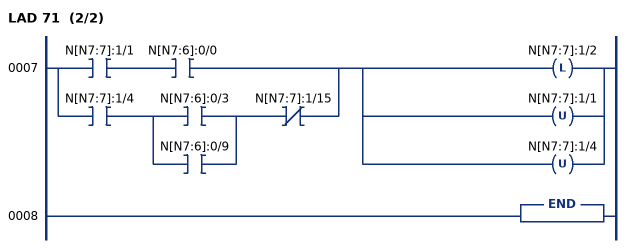
% Rung: 7 %
SOR BST XIC N[N7:7]:1/1 XIC N[N7:6]:0/0 NXB XIC N[N7:7]:1/4 BST XIC N[N7:6]:0/3 NXB XIC N[N7:6]:0/9 BND XIO N[N7:7]:1/15 BND BST OTL N[N7:7]:1/2 NXB OTU N[N7:7]:1/1 NXB OTU N[N7:7]:1/4 BND EOR
% Rung: 8 %
SOR END EOR

LADDER 74
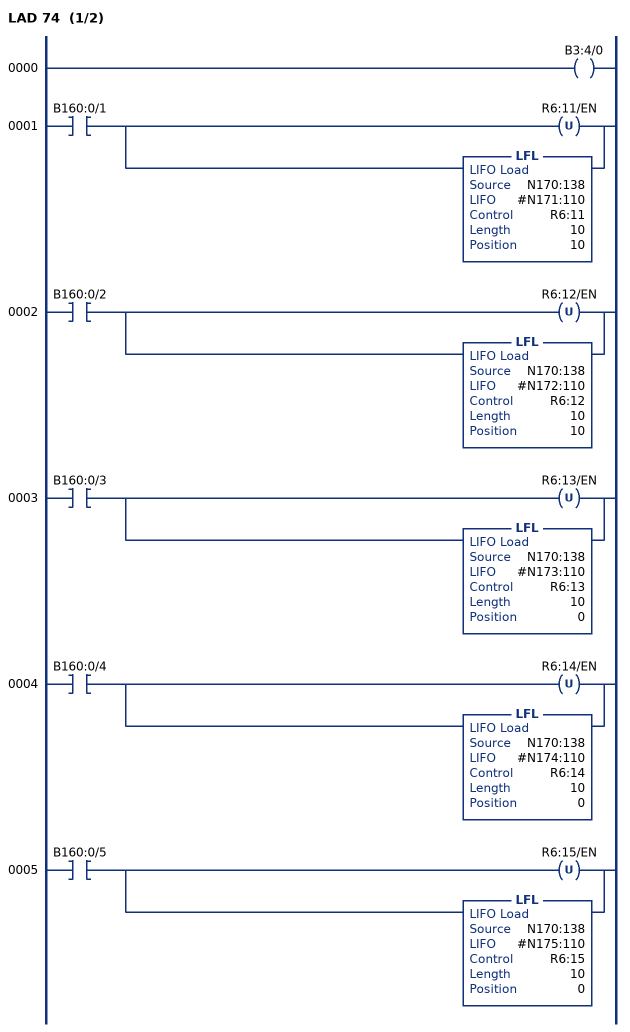
% Rung: 0 %
SOR OTE B3:4/0 EOR
% Rung: 1 %
SOR XIC B160:0/1 BST OTU R6:11/EN NXB LFL N170:138 #N171:110 R6:11 10 10 BND EOR
% Rung: 2 %
SOR XIC B160:0/2 BST OTU R6:12/EN NXB LFL N170:138 #N172:110 R6:12 10 10 BND EOR
% Rung: 3 %
SOR XIC B160:0/3 BST OTU R6:13/EN NXB LFL N170:138 #N173:110 R6:13 10 0 BND EOR
% Rung: 4 %
SOR XIC B160:0/4 BST OTU R6:14/EN NXB LFL N170:138 #N174:110 R6:14 10 0 BND EOR
% Rung: 5 %
SOR XIC B160:0/5 BST OTU R6:15/EN NXB LFL N170:138 #N175:110 R6:15 10 0 BND EOR

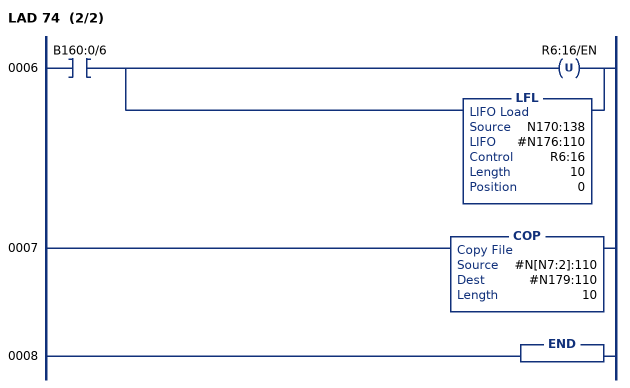
% Rung: 6 %
SOR XIC B160:0/6 BST OTU R6:16/EN NXB LFL N170:138 #N176:110 R6:16 10 0 BND EOR
% Rung: 7 %
SOR COP #N[N7:2]:110 #N179:110 10 EOR
% Rung: 8 %
SOR END EOR

LADDER 75
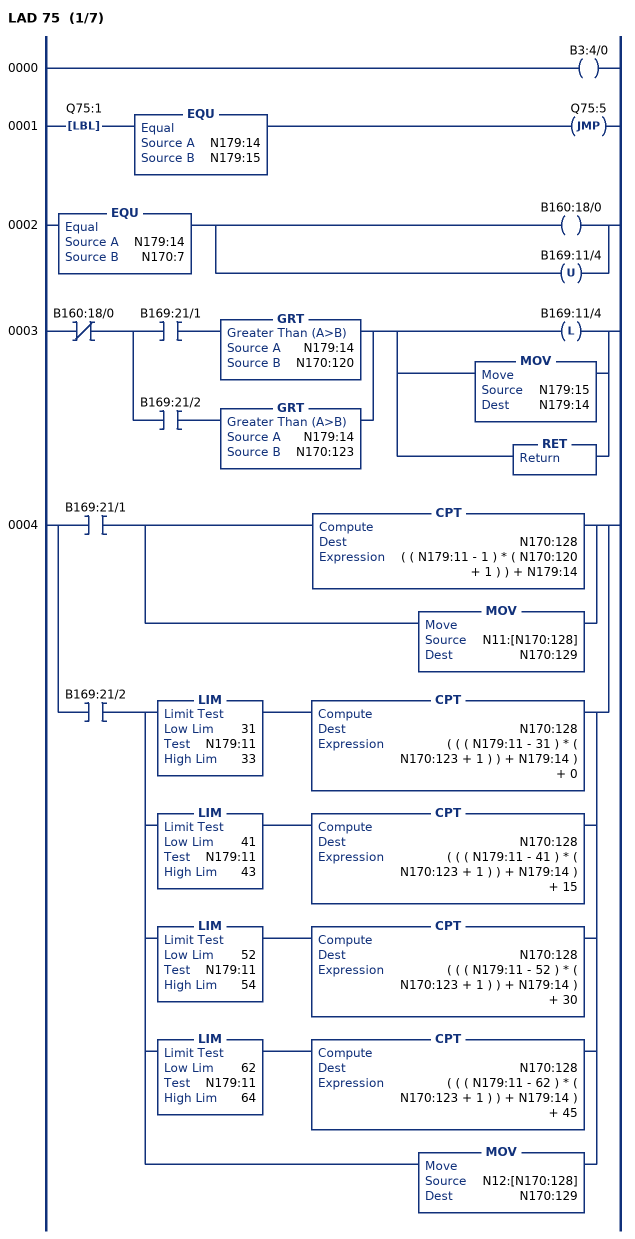
% Rung: 0 %
SOR OTE B3:4/0 EOR
% Rung: 1 %
SOR LBL Q75:1 EQU N179:14 N179:15 JMP Q75:5 EOR
% Rung: 2 %
SOR EQU N179:14 N170:7 BST OTE B160:18/0 NXB OTU B169:11/4 BND EOR
% Rung: 3 %
SOR XIO B160:18/0 BST XIC B169:21/1 GRT N179:14 N170:120 NXB XIC B169:21/2 GRT N179:14 N170:123 BND BST OTL B169:11/4 NXB MOV N179:15 N179:14 NXB RET BND EOR
% Rung: 4 %
SOR BST XIC B169:21/1 BST CPT N170:128 " ( ( N179:11 - 1 ) * ( N170:120 + 1 ) ) + N179:14 " NXB MOV N11:[N170:128] N170:129 BND NXB XIC B169:21/2 BST BST LIM 31 N179:11 33 CPT N170:128 " ( ( ( N179:11 - 31 ) * ( N170:123 + 1 ) ) + N179:14 ) + 0 " NXB LIM 41 N179:11 43 CPT N170:128 " ( ( ( N179:11 - 41 ) * ( N170:123 + 1 ) ) + N179:14 ) + 15 " NXB LIM 52 N179:11 54 CPT N170:128 " ( ( ( N179:11 - 52 ) * ( N170:123 + 1 ) ) + N179:14 ) + 30 " NXB LIM 62 N179:11 64 CPT N170:128 " ( ( ( N179:11 - 62 ) * ( N170:123 + 1 ) ) + N179:14 ) + 45 " BND NXB MOV N12:[N170:128] N170:129 BND BND EOR

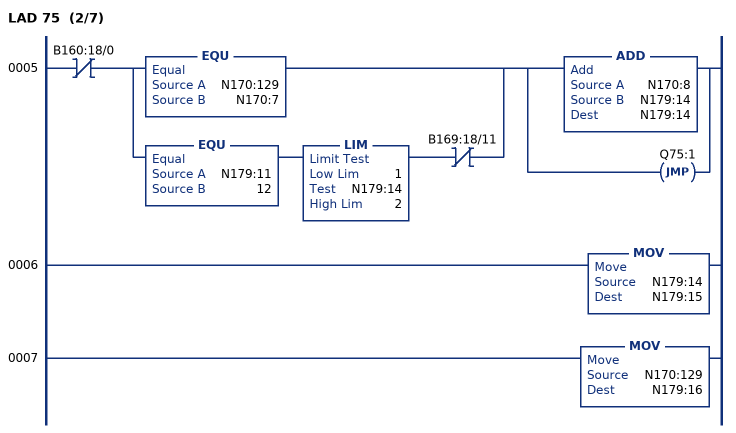
% Rung: 5 %
SOR XIO B160:18/0 BST EQU N170:129 N170:7 NXB EQU N179:11 12 LIM 1 N179:14 2 XIO B169:18/11 BND BST ADD N170:8 N179:14 N179:14 NXB JMP Q75:1 BND EOR
% Rung: 6 %
SOR MOV N179:14 N179:15 EOR
% Rung: 7 %
SOR MOV N170:129 N179:16 EOR

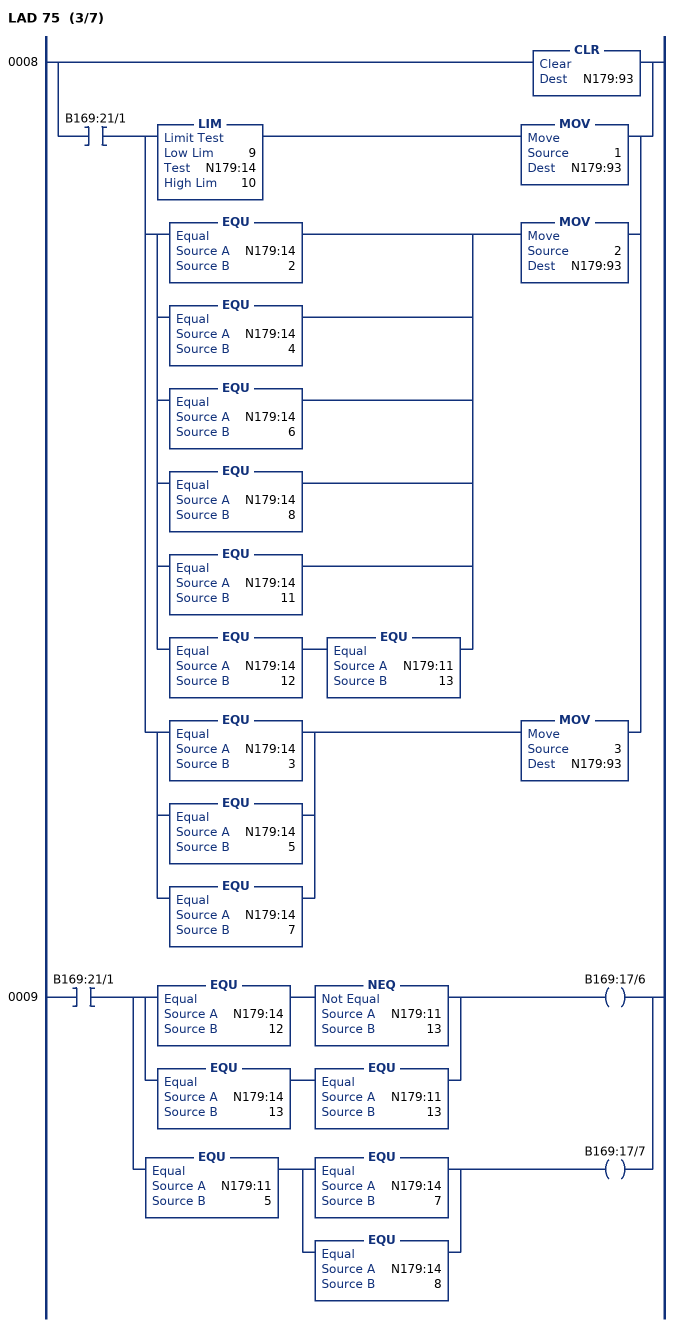
% Rung: 8 %
SOR BST CLR N179:93 NXB XIC B169:21/1 BST LIM 9 N179:14 10 MOV 1 N179:93 NXB BST EQU N179:14 2 NXB EQU N179:14 4 NXB EQU N179:14 6 NXB EQU N179:14 8 NXB EQU N179:14 11 NXB EQU N179:14 12 EQU N179:11 13 BND MOV 2 N179:93 NXB BST EQU N179:14 3 NXB EQU N179:14 5 NXB EQU N179:14 7 BND MOV 3 N179:93 BND BND EOR
% Rung: 9 %
SOR XIC B169:21/1 BST BST EQU N179:14 12 NEQ N179:11 13 NXB EQU N179:14 13 EQU N179:11 13 BND OTE B169:17/6 NXB EQU N179:11 5 BST EQU N179:14 7 NXB EQU N179:14 8 BND OTE B169:17/7 BND EOR

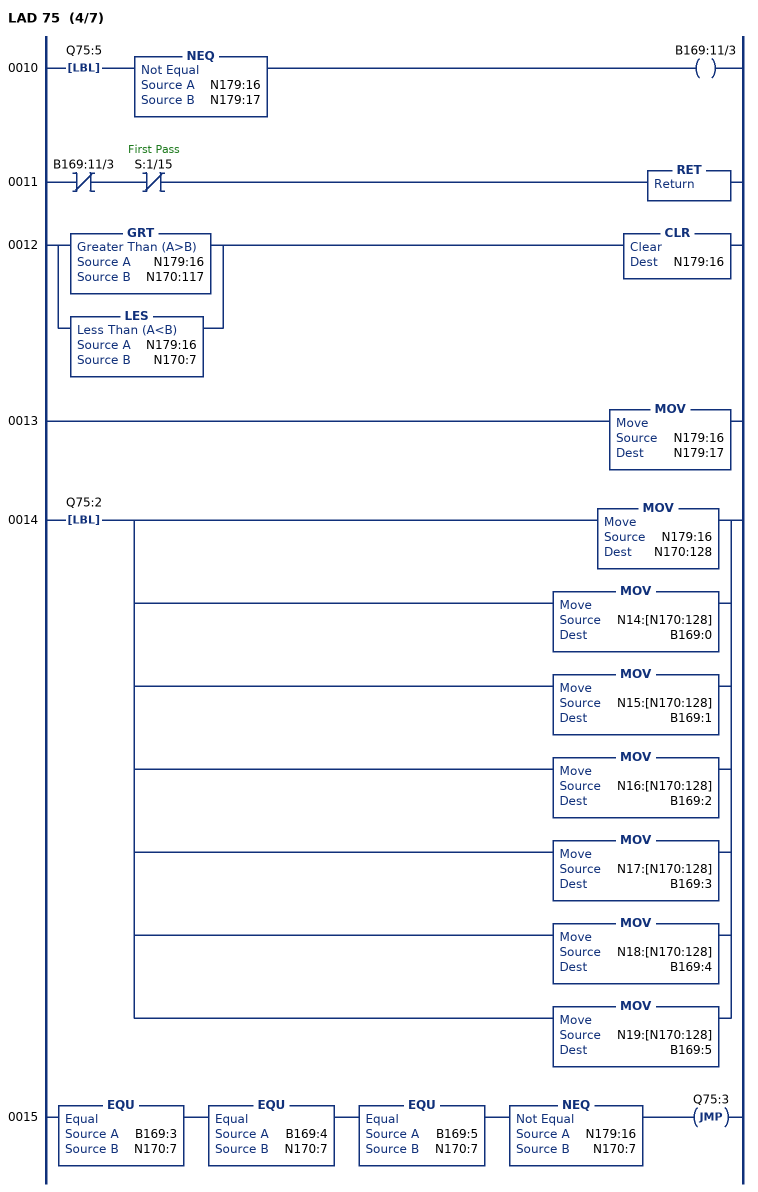
% Rung: 10 %
SOR LBL Q75:5 NEQ N179:16 N179:17 OTE B169:11/3 EOR
% Rung: 11 %
SOR XIO B169:11/3 XIO S:1/15 RET EOR
%   S:1/15  "First Pass" %
% Rung: 12 %
SOR BST GRT N179:16 N170:117 NXB LES N179:16 N170:7 BND CLR N179:16 EOR
% Rung: 13 %
SOR MOV N179:16 N179:17 EOR
% Rung: 14 %
SOR LBL Q75:2 BST MOV N179:16 N170:128 NXB MOV N14:[N170:128] B169:0 NXB MOV N15:[N170:128] B169:1 NXB MOV N16:[N170:128] B169:2 NXB MOV N17:[N170:128] B169:3 NXB MOV N18:[N170:128] B169:4 NXB MOV N19:[N170:128] B169:5 BND EOR
% Rung: 15 %
SOR EQU B169:3 N170:7 EQU B169:4 N170:7 EQU B169:5 N170:7 NEQ N179:16 N170:7 JMP Q75:3 EOR

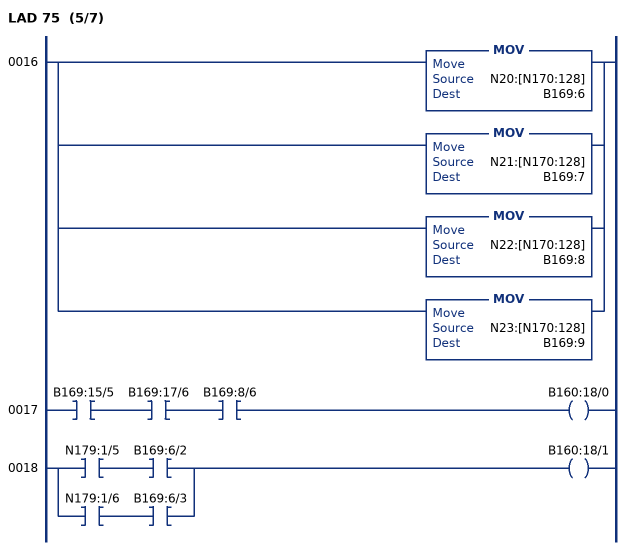
% Rung: 16 %
SOR BST MOV N20:[N170:128] B169:6 NXB MOV N21:[N170:128] B169:7 NXB MOV N22:[N170:128] B169:8 NXB MOV N23:[N170:128] B169:9 BND EOR
% Rung: 17 %
SOR XIC B169:15/5 XIC B169:17/6 XIC B169:8/6 OTE B160:18/0 EOR
% Rung: 18 %
SOR BST XIC N179:1/5 XIC B169:6/2 NXB XIC N179:1/6 XIC B169:6/3 BND OTE B160:18/1 EOR

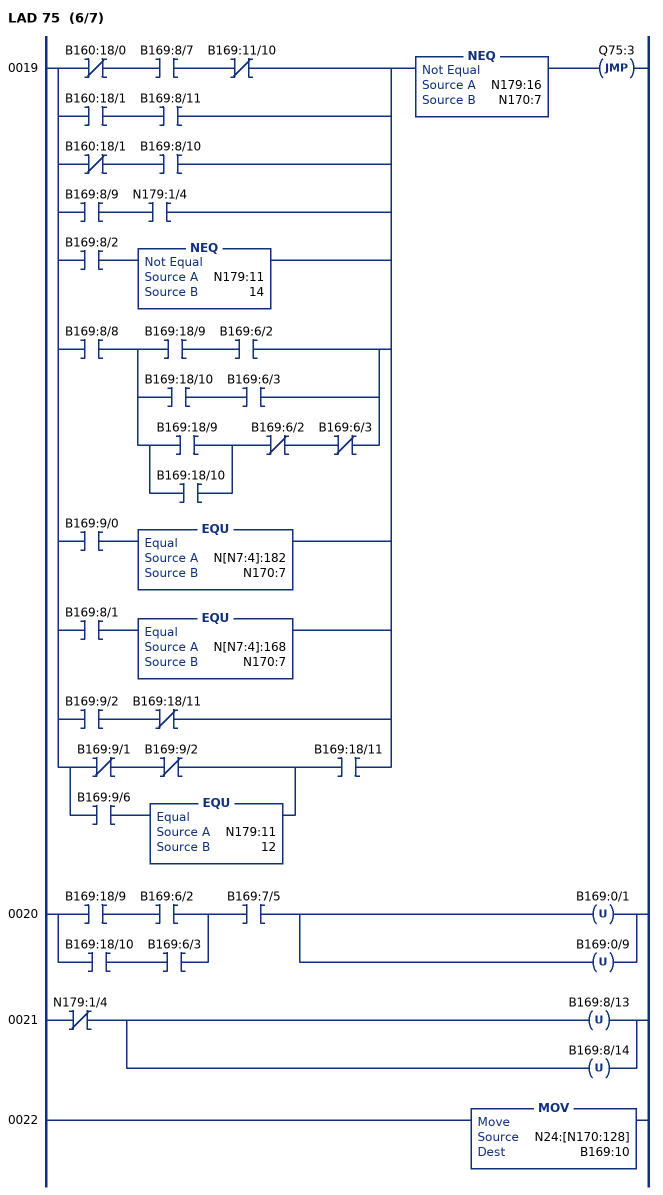
% Rung: 19 %
SOR BST XIO B160:18/0 XIC B169:8/7 XIO B169:11/10 NXB XIC B160:18/1 XIC B169:8/11 NXB XIO B160:18/1 XIC B169:8/10 NXB XIC B169:8/9 XIC N179:1/4 NXB XIC B169:8/2 NEQ N179:11 14 NXB XIC B169:8/8 BST XIC B169:18/9 XIC B169:6/2 NXB XIC B169:18/10 XIC B169:6/3 NXB BST XIC B169:18/9 NXB XIC B169:18/10 BND XIO B169:6/2 XIO B169:6/3 BND NXB XIC B169:9/0 EQU N[N7:4]:182 N170:7 NXB XIC B169:8/1 EQU N[N7:4]:168 N170:7 NXB XIC B169:9/2 XIO B169:18/11 NXB BST XIO B169:9/1 XIO B169:9/2 NXB XIC B169:9/6 EQU N179:11 12 BND XIC B169:18/11 BND NEQ N179:16 N170:7 JMP Q75:3 EOR
% Rung: 20 %
SOR BST XIC B169:18/9 XIC B169:6/2 NXB XIC B169:18/10 XIC B169:6/3 BND XIC B169:7/5 BST OTU B169:0/1 NXB OTU B169:0/9 BND EOR
% Rung: 21 %
SOR XIO N179:1/4 BST OTU B169:8/13 NXB OTU B169:8/14 BND EOR
% Rung: 22 %
SOR MOV N24:[N170:128] B169:10 EOR

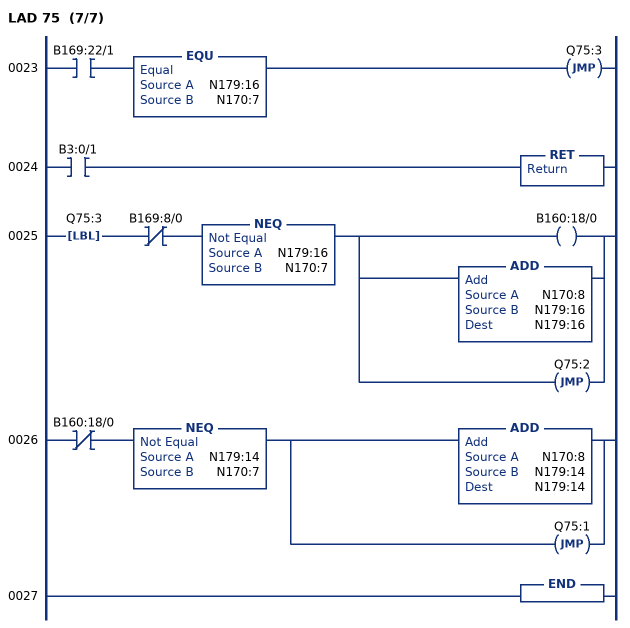
% Rung: 23 %
SOR XIC B169:22/1 EQU N179:16 N170:7 JMP Q75:3 EOR
% Rung: 24 %
SOR XIC B3:0/1 RET EOR
% Rung: 25 %
SOR LBL Q75:3 XIO B169:8/0 NEQ N179:16 N170:7 BST OTE B160:18/0 NXB ADD N170:8 N179:16 N179:16 NXB JMP Q75:2 BND EOR
% Rung: 26 %
SOR XIO B160:18/0 NEQ N179:14 N170:7 BST ADD N170:8 N179:14 N179:14 NXB JMP Q75:1 BND EOR
% Rung: 27 %
SOR END EOR

LADDER 76
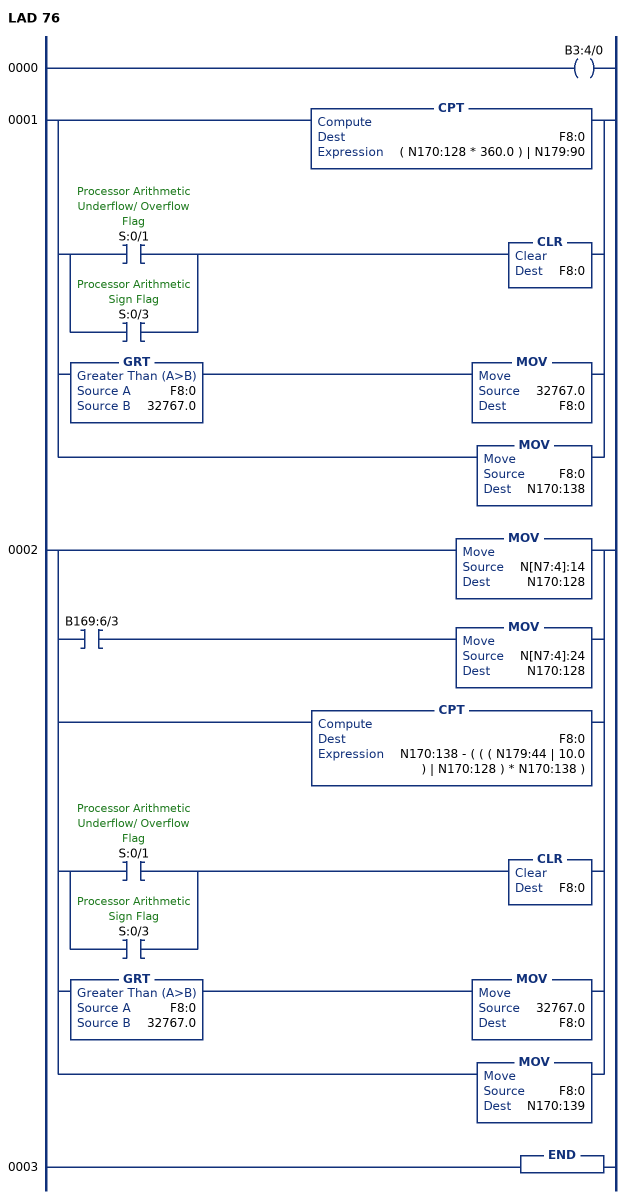
% Rung: 0 %
SOR OTE B3:4/0 EOR
% Rung: 1 %
SOR BST CPT F8:0 " ( N170:128 * 360.0 ) | N179:90 " NXB BST XIC S:0/1 NXB XIC S:0/3 BND CLR F8:0 NXB GRT F8:0 32767.0 MOV 32767.0 F8:0 NXB MOV F8:0 N170:138 BND EOR
%   S:0/1  "Processor Arithmetic Underflow/ Overflow Flag" %
%   S:0/3  "Processor Arithmetic Sign Flag" %
% Rung: 2 %
SOR BST MOV N[N7:4]:14 N170:128 NXB XIC B169:6/3 MOV N[N7:4]:24 N170:128 NXB CPT F8:0 " N170:138 - ( ( ( N179:44 | 10.0 ) | N170:128 ) * N170:138 ) " NXB BST XIC S:0/1 NXB XIC S:0/3 BND CLR F8:0 NXB GRT F8:0 32767.0 MOV 32767.0 F8:0 NXB MOV F8:0 N170:139 BND EOR
%   S:0/1  "Processor Arithmetic Underflow/ Overflow Flag" %
%   S:0/3  "Processor Arithmetic Sign Flag" %
% Rung: 3 %
SOR END EOR

LADDER 77
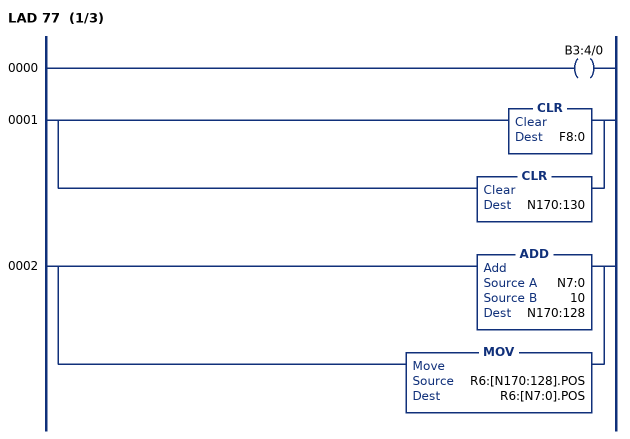
% Rung: 0 %
SOR OTE B3:4/0 EOR
% Rung: 1 %
SOR BST CLR F8:0 NXB CLR N170:130 BND EOR
% Rung: 2 %
SOR BST ADD N7:0 10 N170:128 NXB MOV R6:[N170:128].POS R6:[N7:0].POS BND EOR

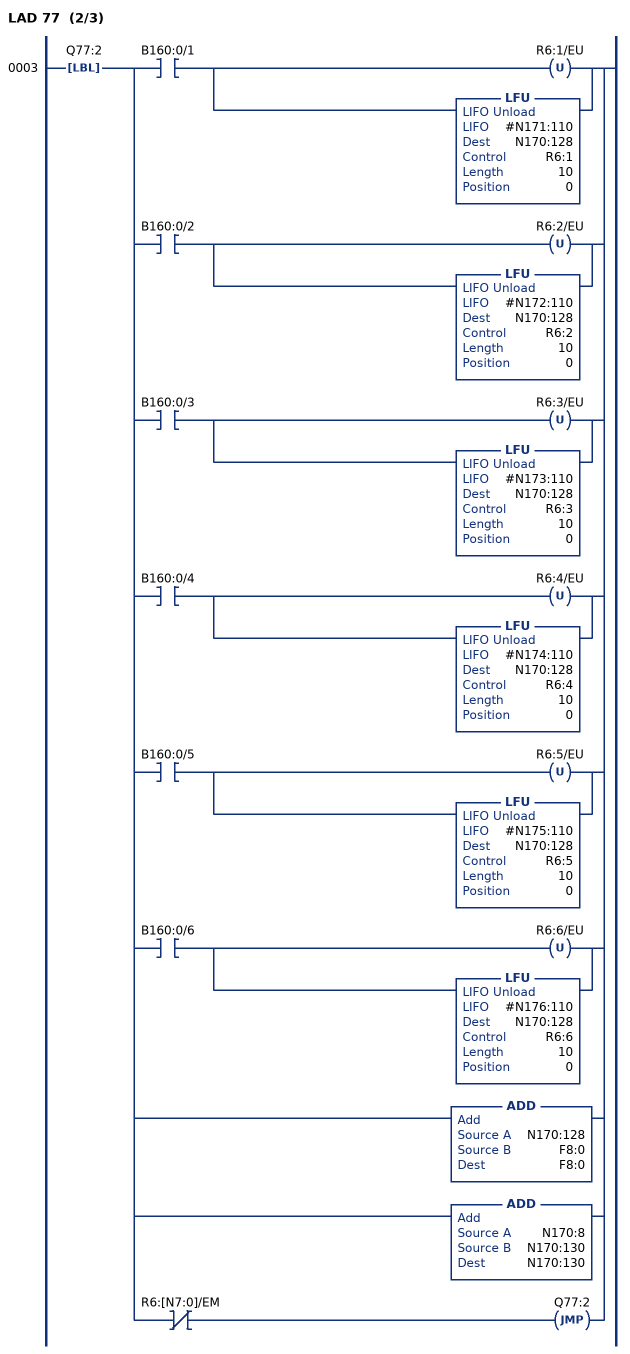
% Rung: 3 %
SOR LBL Q77:2 BST XIC B160:0/1 BST OTU R6:1/EU NXB LFU #N171:110 N170:128 R6:1 10 0 BND NXB XIC B160:0/2 BST OTU R6:2/EU NXB LFU #N172:110 N170:128 R6:2 10 0 BND NXB XIC B160:0/3 BST OTU R6:3/EU NXB LFU #N173:110 N170:128 R6:3 10 0 BND NXB XIC B160:0/4 BST OTU R6:4/EU NXB LFU #N174:110 N170:128 R6:4 10 0 BND NXB XIC B160:0/5 BST OTU R6:5/EU NXB LFU #N175:110 N170:128 R6:5 10 0 BND NXB XIC B160:0/6 BST OTU R6:6/EU NXB LFU #N176:110 N170:128 R6:6 10 0 BND NXB ADD N170:128 F8:0 F8:0 NXB ADD N170:8 N170:130 N170:130 NXB XIO R6:[N7:0]/EM JMP Q77:2 BND EOR

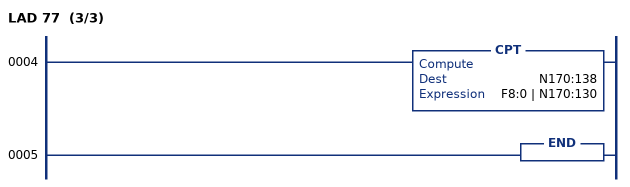
% Rung: 4 %
SOR CPT N170:138 " F8:0 | N170:130 " EOR
% Rung: 5 %
SOR END EOR

LADDER 78
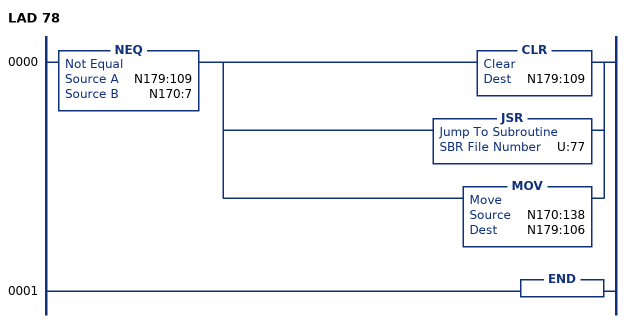
% Rung: 0 %
SOR NEQ N179:109 N170:7 BST CLR N179:109 NXB JSR U:77 NXB MOV N170:138 N179:106 BND EOR
% Rung: 1 %
SOR END EOR

LADDER 79
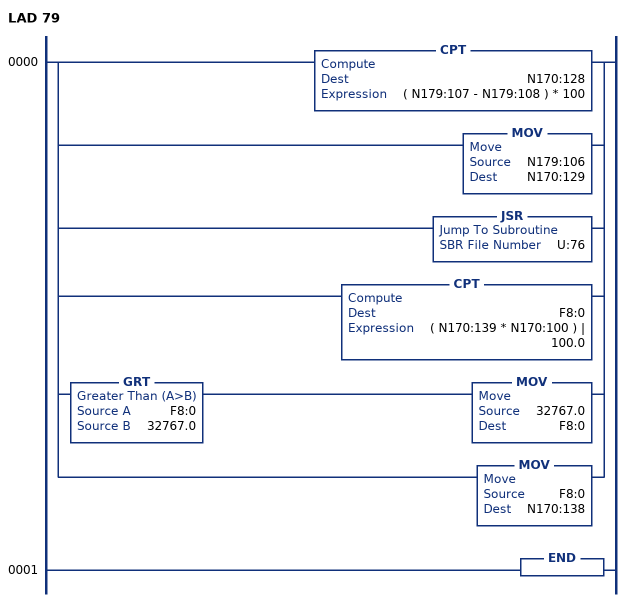
% Rung: 0 %
SOR BST CPT N170:128 " ( N179:107 - N179:108 ) * 100 " NXB MOV N179:106 N170:129 NXB JSR U:76 NXB CPT F8:0 " ( N170:139 * N170:100 ) | 100.0 " NXB GRT F8:0 32767.0 MOV 32767.0 F8:0 NXB MOV F8:0 N170:138 BND EOR
% Rung: 1 %
SOR END EOR

LADDER 80
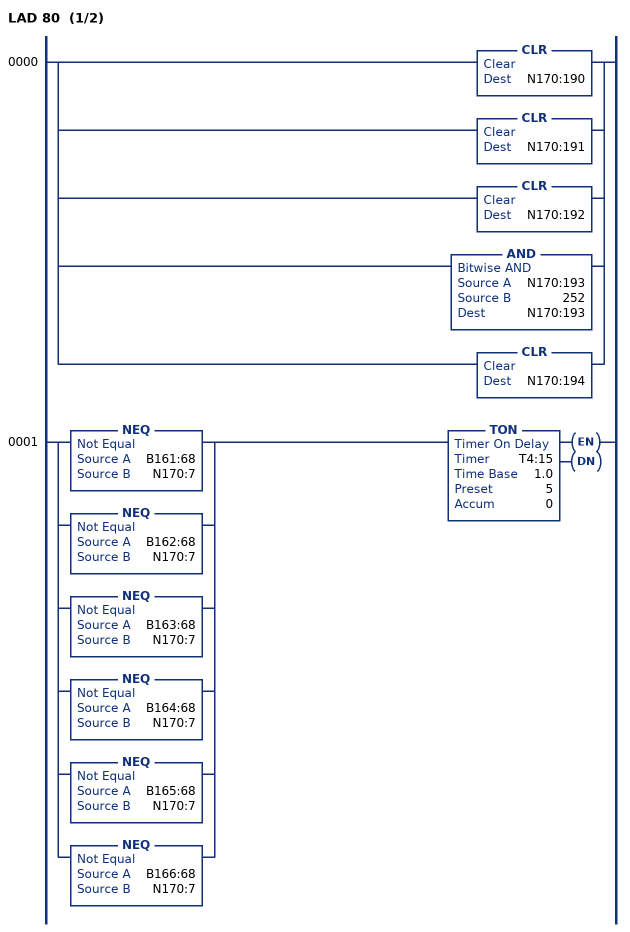
% Rung: 0 %
SOR BST CLR N170:190 NXB CLR N170:191 NXB CLR N170:192 NXB AND N170:193 252 N170:193 NXB CLR N170:194 BND EOR
% Rung: 1 %
SOR BST NEQ B161:68 N170:7 NXB NEQ B162:68 N170:7 NXB NEQ B163:68 N170:7 NXB NEQ B164:68 N170:7 NXB NEQ B165:68 N170:7 NXB NEQ B166:68 N170:7 BND TON T4:15 1.0 5 0 EOR

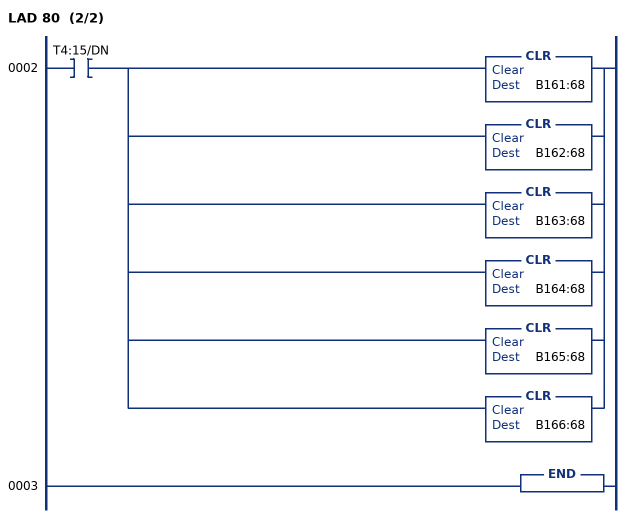
% Rung: 2 %
SOR XIC T4:15/DN BST CLR B161:68 NXB CLR B162:68 NXB CLR B163:68 NXB CLR B164:68 NXB CLR B165:68 NXB CLR B166:68 BND EOR
% Rung: 3 %
SOR END EOR

LADDER 81
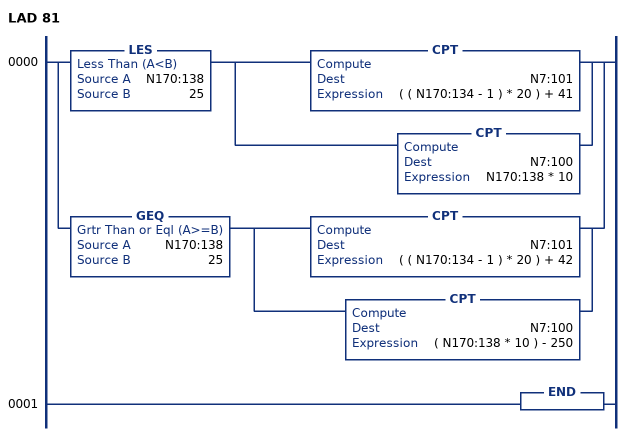
% Rung: 0 %
SOR BST LES N170:138 25 BST CPT N7:101 " ( ( N170:134 - 1 ) * 20 ) + 41 " NXB CPT N7:100 " N170:138 * 10 " BND NXB GEQ N170:138 25 BST CPT N7:101 " ( ( N170:134 - 1 ) * 20 ) + 42 " NXB CPT N7:100 " ( N170:138 * 10 ) - 250 " BND BND EOR
% Rung: 1 %
SOR END EOR

LADDER 82
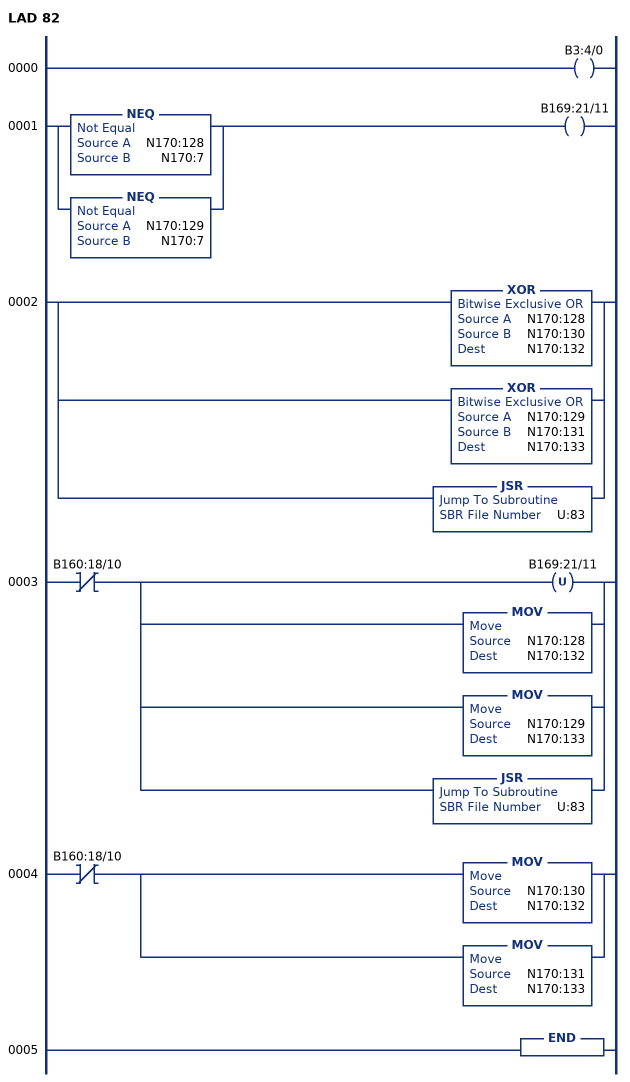
% Rung: 0 %
SOR OTE B3:4/0 EOR
% Rung: 1 %
SOR BST NEQ N170:128 N170:7 NXB NEQ N170:129 N170:7 BND OTE B169:21/11 EOR
% Rung: 2 %
SOR BST XOR N170:128 N170:130 N170:132 NXB XOR N170:129 N170:131 N170:133 NXB JSR U:83 BND EOR
% Rung: 3 %
SOR XIO B160:18/10 BST OTU B169:21/11 NXB MOV N170:128 N170:132 NXB MOV N170:129 N170:133 NXB JSR U:83 BND EOR
% Rung: 4 %
SOR XIO B160:18/10 BST MOV N170:130 N170:132 NXB MOV N170:131 N170:133 BND EOR
% Rung: 5 %
SOR END EOR

LADDER 83
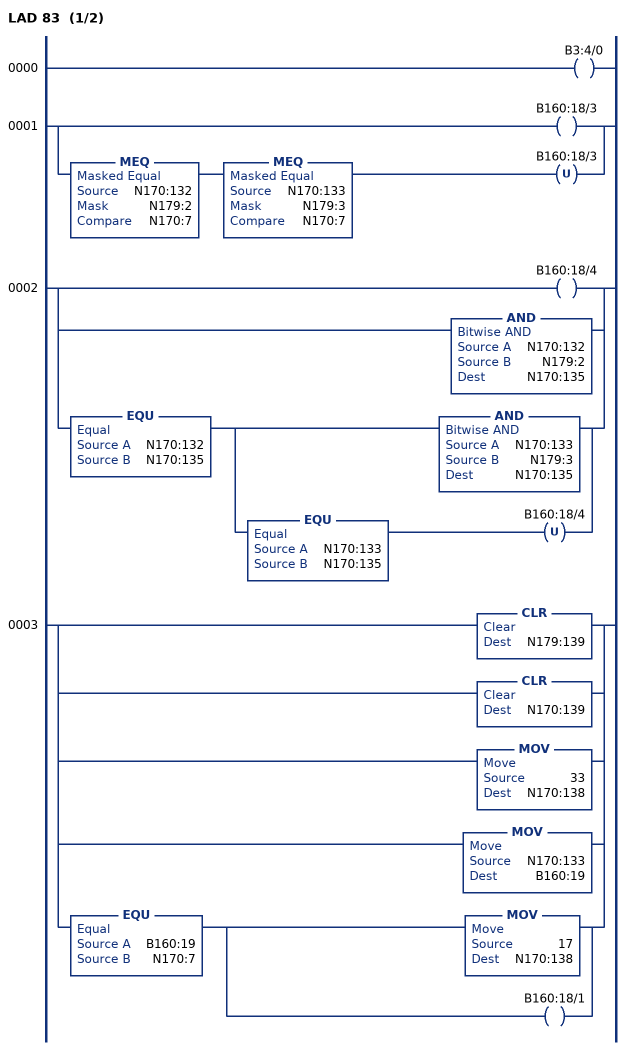
% Rung: 0 %
SOR OTE B3:4/0 EOR
% Rung: 1 %
SOR BST OTE B160:18/3 NXB MEQ N170:132 N179:2 N170:7 MEQ N170:133 N179:3 N170:7 OTU B160:18/3 BND EOR
% Rung: 2 %
SOR BST OTE B160:18/4 NXB AND N170:132 N179:2 N170:135 NXB EQU N170:132 N170:135 BST AND N170:133 N179:3 N170:135 NXB EQU N170:133 N170:135 OTU B160:18/4 BND BND EOR
% Rung: 3 %
SOR BST CLR N179:139 NXB CLR N170:139 NXB MOV 33 N170:138 NXB MOV N170:133 B160:19 NXB EQU B160:19 N170:7 BST MOV 17 N170:138 NXB OTE B160:18/1 BND BND EOR

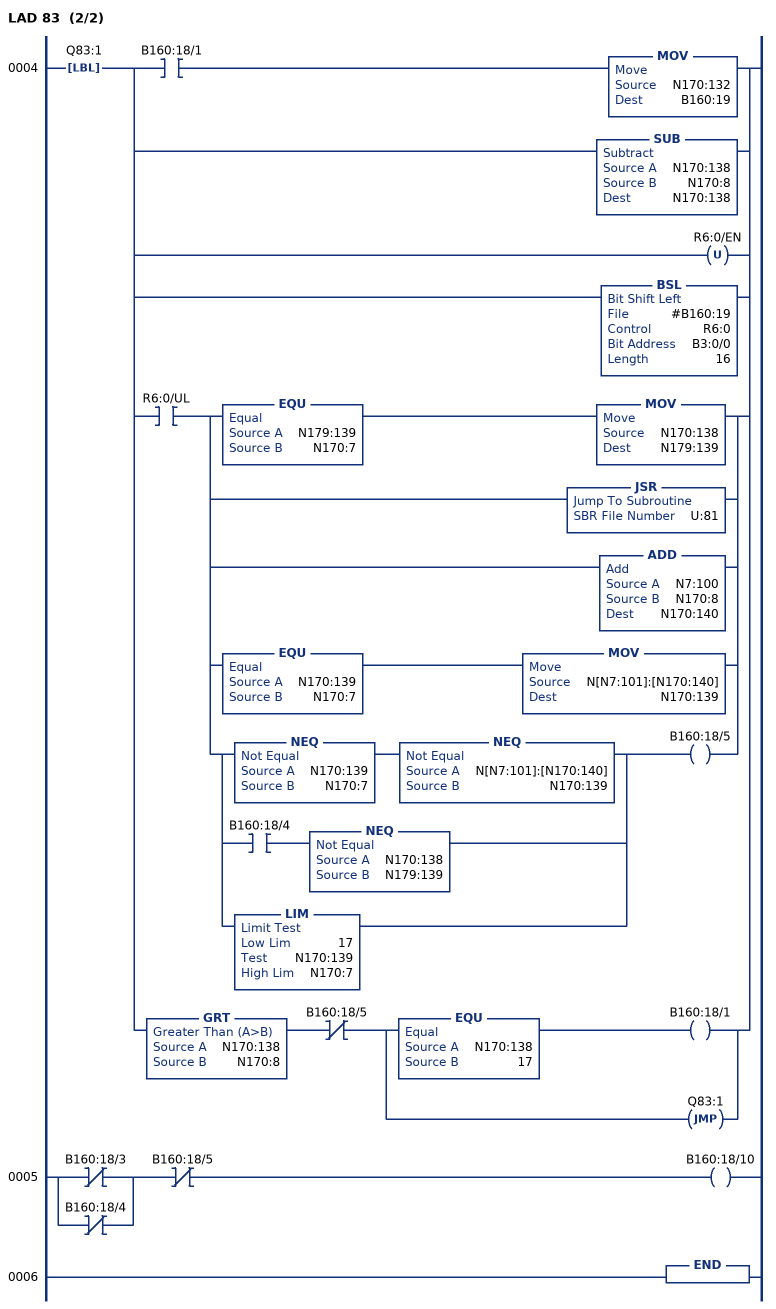
% Rung: 4 %
SOR LBL Q83:1 BST XIC B160:18/1 MOV N170:132 B160:19 NXB SUB N170:138 N170:8 N170:138 NXB OTU R6:0/EN NXB BSL #B160:19 R6:0 B3:0/0 16 NXB XIC R6:0/UL BST EQU N179:139 N170:7 MOV N170:138 N179:139 NXB JSR U:81 NXB ADD N7:100 N170:8 N170:140 NXB EQU N170:139 N170:7 MOV N[N7:101]:[N170:140] N170:139 NXB BST NEQ N170:139 N170:7 NEQ N[N7:101]:[N170:140] N170:139 NXB XIC B160:18/4 NEQ N170:138 N179:139 NXB LIM 17 N170:139 N170:7 BND OTE B160:18/5 BND NXB GRT N170:138 N170:8 XIO B160:18/5 BST EQU N170:138 17 OTE B160:18/1 NXB JMP Q83:1 BND BND EOR
% Rung: 5 %
SOR BST XIO B160:18/3 NXB XIO B160:18/4 BND XIO B160:18/5 OTE B160:18/10 EOR
% Rung: 6 %
SOR END EOR

LADDER 101
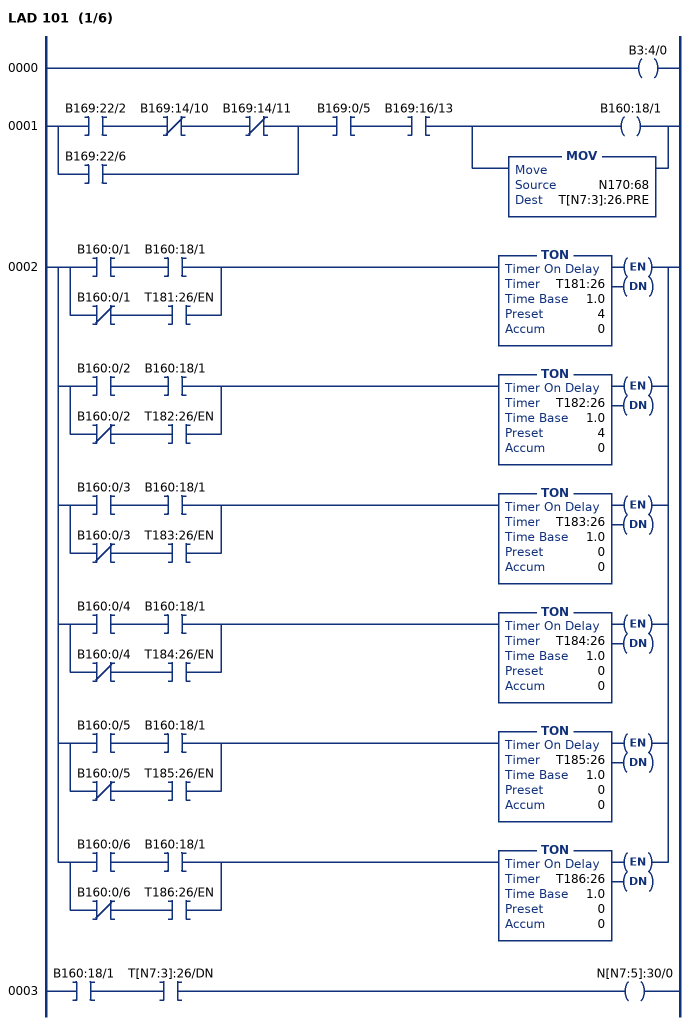
% Rung: 0 %
SOR OTE B3:4/0 EOR
% Rung: 1 %
SOR BST XIC B169:22/2 XIO B169:14/10 XIO B169:14/11 NXB XIC B169:22/6 BND XIC B169:0/5 XIC B169:16/13 BST OTE B160:18/1 NXB MOV N170:68 T[N7:3]:26.PRE BND EOR
% Rung: 2 %
SOR BST BST XIC B160:0/1 XIC B160:18/1 NXB XIO B160:0/1 XIC T181:26/EN BND TON T181:26 1.0 4 0 NXB BST XIC B160:0/2 XIC B160:18/1 NXB XIO B160:0/2 XIC T182:26/EN BND TON T182:26 1.0 4 0 NXB BST XIC B160:0/3 XIC B160:18/1 NXB XIO B160:0/3 XIC T183:26/EN BND TON T183:26 1.0 0 0 NXB BST XIC B160:0/4 XIC B160:18/1 NXB XIO B160:0/4 XIC T184:26/EN BND TON T184:26 1.0 0 0 NXB BST XIC B160:0/5 XIC B160:18/1 NXB XIO B160:0/5 XIC T185:26/EN BND TON T185:26 1.0 0 0 NXB BST XIC B160:0/6 XIC B160:18/1 NXB XIO B160:0/6 XIC T186:26/EN BND TON T186:26 1.0 0 0 BND EOR
% Rung: 3 %
SOR XIC B160:18/1 XIC T[N7:3]:26/DN OTE N[N7:5]:30/0 EOR

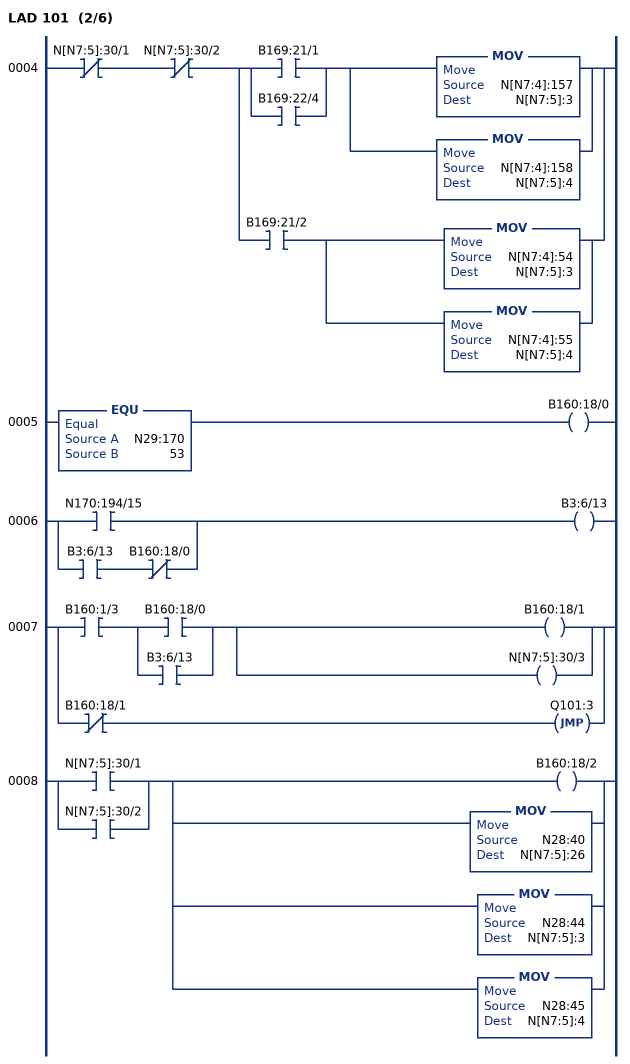
% Rung: 4 %
SOR XIO N[N7:5]:30/1 XIO N[N7:5]:30/2 BST BST XIC B169:21/1 NXB XIC B169:22/4 BND BST MOV N[N7:4]:157 N[N7:5]:3 NXB MOV N[N7:4]:158 N[N7:5]:4 BND NXB XIC B169:21/2 BST MOV N[N7:4]:54 N[N7:5]:3 NXB MOV N[N7:4]:55 N[N7:5]:4 BND BND EOR
% Rung: 5 %
SOR EQU N29:170 53 OTE B160:18/0 EOR
% Rung: 6 %
SOR BST XIC N170:194/15 NXB XIC B3:6/13 XIO B160:18/0 BND OTE B3:6/13 EOR
% Rung: 7 %
SOR BST XIC B160:1/3 BST XIC B160:18/0 NXB XIC B3:6/13 BND BST OTE B160:18/1 NXB OTE N[N7:5]:30/3 BND NXB XIO B160:18/1 JMP Q101:3 BND EOR
% Rung: 8 %
SOR BST XIC N[N7:5]:30/1 NXB XIC N[N7:5]:30/2 BND BST OTE B160:18/2 NXB MOV N28:40 N[N7:5]:26 NXB MOV N28:44 N[N7:5]:3 NXB MOV N28:45 N[N7:5]:4 BND EOR

